ABB RobotStudio station: gripper.rsstn

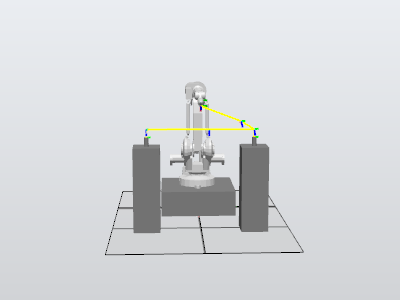
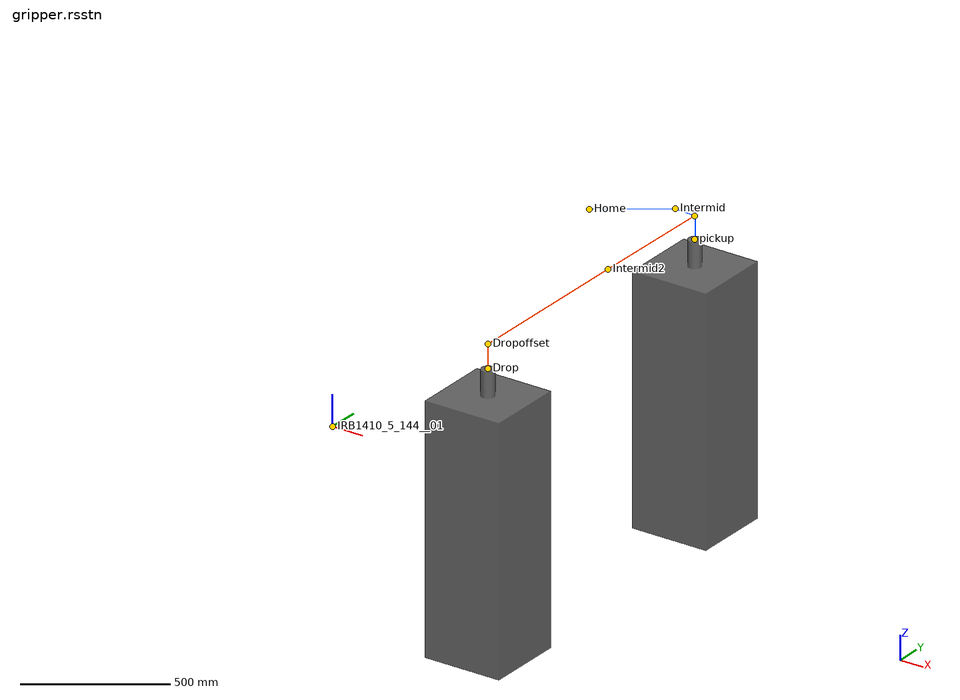
[picture v1: parts stored in the station drawn from their meshes, with robot base, taught points and paths (robot models come from the ABB library and are not in the file)]
Station Station (saved by RobotStudio 22.3.10141.1)
Controller IRB1410, task T_ROB1: task frame (RAPID world) sits at (0, 0, 300) mm in the station
Controller IRB1410
  mechanical unit ROB_1: IRB1410_5_144__01, 6 joints, base frame (0, 0, 0) mm
Layout (positions relative to the parent item):
  - IRB1410_5_144__01 [mechanism, from Robots\IRB1410_5_144_G_01.rslib] at (0, 0, 300) mm; joint values [0, 0, 0, 0, 0.5236, 0] (rad or m)
  - concrete [part, from Dispencing\Concrete.rslib] at (-450, -450, 0) mm
  - Part_1 [part] at (1800, 1050, 0) mm, size 300 x 300 x 950 mm
  - Part_2 [part] at (1053.15, 595.29, 950) mm, size 50 x 49.9 x 100 mm
  - Part_3 [part] at (1053.15, -604.71, 950) mm, size 50 x 49.9 x 100 mm
  - Part_4 [part] at (1800, -150, 0) mm, size 300 x 300 x 950 mm
  - SmartComponent_1 [smart component]
      signals: DI close
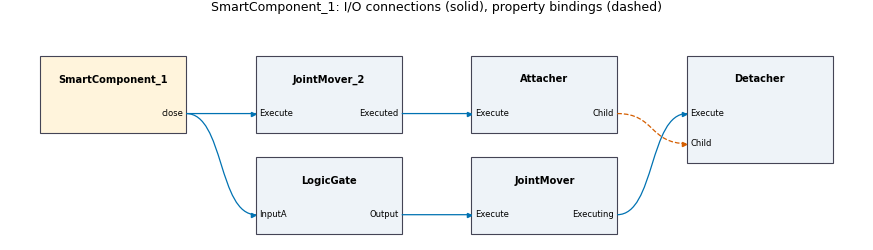
      connections:
        JointMover_2.Executed -> Attacher.Execute
        JointMover.Executing -> Detacher.Execute
        SmartComponent_1.close -> JointMover_2.Execute
        SmartComponent_1.close -> LogicGate.InputA
        LogicGate.Output -> JointMover.Execute
        Attacher.Child => Detacher.Child
    - JointMover [smart component, from Components\JointMover.rslib]
        properties: Mechanism=Smart_Gripper_Servo_Fingers; Relative=false; Duration=0; J1=0.025
    - JointMover_2 [smart component, from Components\JointMover.rslib]
        properties: Mechanism=Smart_Gripper_Servo_Fingers; Relative=false; Duration=0; J1=0.024
    - Attacher [smart component, from Components\Attacher.rslib]
        properties: Parent=Smart_Gripper_Servo_Fingers; Flange=0; Child=Part_2; Mount=false; Offset=[0 0 0]; Orientation=[0 0 0]
    - Detacher [smart component, from Components\Detacher.rslib]
        properties: Child=Part_2; KeepPosition=true
    - Smart_Gripper_Servo_Fingers [mechanism, from Tools\ABB_Smart_Gripper_Servo_Fingers.rslib] at (943.61, 0, 1452.5) mm, rotated rx 180 ry 60 rz 180 deg; joint values [0.025] (rad or m)
    - LogicGate [smart component, from Components\LogicGate.rslib]
        properties: Operator=NOT; Delay=0
Attachment: Smart_Gripper_Servo_Fingers is attached to IRB1410_5_144__01 / Link6
Station logic (signal -> signal, property => property):
  IRB1410.cls -> SmartComponent_1.close
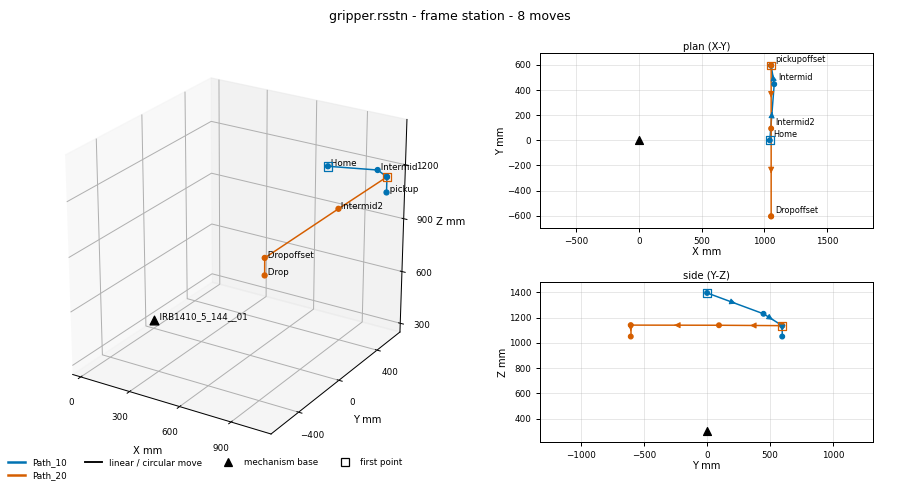
[picture p0: tool path of gripper.rsstn in frame station, 8 of 8 moves have a stored position in this frame; points joined in program order, loops and branches not executed]
Targets, tools, work objects and paths stored in the station, written as RAPID:
! task T_ROB1
MODULE CalibData
  PERS tooldata Servo:=[TRUE,[[0,0,114.2],[1,0,0,0]],[0.215,[8.7,12.3,49.2],[1,0,0,0],0.00021,0.00024,0.00009]];
ENDMODULE

! task T_ROB1
MODULE Module1
  CONST robtarget Home:=[[1042.512260434,0,1095.4],[0.5,0,0.866025404,0],[0,0,0,0],[9E+09,9E+09,9E+09,9E+09,9E+09,9E+09]];
  CONST robtarget Intermid:=[[1077.460969638,446.838090231,930.152405502],[0.245074316,-0.129670398,0.959483632,0.050153041],[0,-1,0,0],[9E+09,9E+09,9E+09,9E+09,9E+09,9E+09]];
  CONST robtarget pickupoffset:=[[1053.146916662,595.291900705,836.173709095],[0.052986024,-0.016951858,0.995965221,0.070415872],[0,0,0,0],[9E+09,9E+09,9E+09,9E+09,9E+09,9E+09]];
  CONST robtarget pickup:=[[1053.150045291,595.289971364,749.999989829],[0.000019949,-0.020767908,0.999783863,-0.000959717],[0,-1,0,0],[9E+09,9E+09,9E+09,9E+09,9E+09,9E+09]];
  CONST robtarget Intermid2:=[[1053.150026505,94.179124131,839.394204715],[0.000019933,-0.020767891,0.999783863,-0.000959717],[0,-1,0,0],[9E+09,9E+09,9E+09,9E+09,9E+09,9E+09]];
  CONST robtarget Drop:=[[1053.146922276,-604.708049939,749.999578133],[0.000019947,-0.020767907,0.999783863,-0.000959726],[-1,-1,-1,0],[9E+09,9E+09,9E+09,9E+09,9E+09,9E+09]];
  CONST robtarget Dropoffset:=[[1053.146920631,-604.708048994,840.560067009],[0.000019931,-0.020767893,0.999783863,-0.000959716],[-1,-1,-1,0],[9E+09,9E+09,9E+09,9E+09,9E+09,9E+09]];
  PROC Path_10()
    MoveL Home,v1000,z100,Servo\WObj:=wobj0;
    MoveL Intermid,v1000,z100,Servo\WObj:=wobj0;
    MoveL pickupoffset,v1000,z100,Servo\WObj:=wobj0;
    MoveL pickup,v1000,z100,Servo\WObj:=wobj0;
    WaitTime 1;
    SetDO cls,1;
  ENDPROC
  PROC Path_20()
    MoveL pickupoffset,v1000,z100,Servo\WObj:=wobj0;
    MoveL Intermid2,v1000,z100,Servo\WObj:=wobj0;
    MoveL Dropoffset,v1000,z100,Servo\WObj:=wobj0;
    MoveL Drop,v1000,z100,Servo\WObj:=wobj0;
    WaitTime 1;
    SetDO cls,0;
  ENDPROC
  PROC Path_30()
    Path_10;
    Path_20;
  ENDPROC
ENDMODULE

